{attribute 'linkalways'} 
{attribute 'no_explicit_call' := 'This FB is a CLASS and must be accessed using methods or properties'}
FUNCTION_BLOCK Nci EXTENDS CyclicInstance IMPLEMENTS I_Nci
VAR
	_nciPlc : NciPlc;
END_VAR

PROPERTY _InternalNciPlcRef : REFERENCE TO NciPlc
GET
_InternalNciPlcRef REF= _nciPlc;
END_GET
END_PROPERTY

METHOD AddAxisToGroup
VAR_INPUT
	axis : I_Axis;
	index : UDINT;
	timeout : TIME;
	feedback : REFERENCE TO I_CommandFeedback;
END_VAR
VAR_INST
	pCmd : POINTER TO AddAxisToGroupCommand;
END_VAR
VAR
	_axis : I_Axis;
	_index : UDINT;
	_timeout : TIME;
END_VAR
_axis := axis;
_index := index;
_timeout := timeout;

pCmd := __NEW(AddAxisToGroupCommand(
	nci := THIS^,
	axis := _axis,
	index := _index,
	timeout := _timeout
));

(*
This doesn't work hence the horrible hack with intermediate values

pCmd := __NEW(AddAxisToGroupCommand(
	nci := THIS^,
	axis := axis,
	index := index,
	timeout := timeout
));
*)

pCmd^.Execute(feedback).ThenRelease();
END_METHOD

PROPERTY BlockNumber : UDINT
GET
BlockNumber := ItpGetBlockNumber(THIS^._nciPlc.nciToPlc);
END_GET
END_PROPERTY

METHOD BuildXYGroup
VAR_INPUT
	xAxis : I_Axis;
	yAxis : I_Axis;
	timeout : TIME;
	feedback : REFERENCE TO I_CommandFeedback;
END_VAR
VAR
	null : I_Axis;
END_VAR
BuildXYZGroup(xAxis, yAxis, null, timeout, feedback);
END_METHOD

METHOD BuildXYZGroup
VAR_INPUT
	xAxis : I_Axis;
	yAxis : I_Axis;
	zAxis : I_Axis;
	timeout : TIME;
	feedback : REFERENCE TO I_CommandFeedback;
END_VAR
VAR_INST
	pCmd : POINTER TO BuildXYZGroupCommand;
END_VAR
VAR
	_xAxis : I_Axis;
	_yAxis : I_Axis;
	_zAxis : I_Axis;
	_timeout : TIME;
END_VAR
_xAxis := xAxis;
_yAxis := yAxis;
_zAxis := zAxis;
_timeout := timeout;

pCmd := __NEW(BuildXYZGroupCommand(
	nci := THIS^,
	xAxis := _xAxis,
	yAxis := _yAxis,
	zAxis := _zAxis,
	timeout := _timeout
));

(*
This doesn't work hence the horrible hack with intermediate values

pCmd := __NEW(BuildXYZGroupCommand(
	nci := THIS^,
	xAxis := xAxis,
	yAxis := yAxis,
	zAxis := zAxis,
	timeout := commandTimeout
));
*)

pCmd^.Execute(feedback).ThenRelease();
END_METHOD

PROPERTY ChannelId : UINT
GET
ChannelId := ItpGetChannelId(THIS^._nciPlc.nciToPlc);
END_GET
END_PROPERTY

PROPERTY ChannelType : ChannelType
GET
VAR
	inter : INT;
	pInter : POINTER TO ChannelType;
END_VAR
// Don't know how to do the type conversion with NCIChannelType being strict
inter := ItpGetChannelType(THIS^._nciPlc.nciToPlc);
pInter := ADR(inter);
ChannelType := pInter^;
END_GET
END_PROPERTY

METHOD  CyclicCall
END_METHOD

PROPERTY ErrorId : UDINT
GET
ErrorId := ItpGetError(THIS^._nciPlc.nciToPlc);
END_GET
END_PROPERTY

METHOD GetGroupAxisIds : DWORD
VAR_IN_OUT
	axisIds : ARRAY[1..8] OF DWORD;
END_VAR
GetGroupAxisIds := ItpGetGroupAxisIds(axisIds, THIS^._nciPlc.nciToPlc);
END_METHOD

METHOD GetOverride : LREAL
GetOverride := ItpGetOverridePercent(THIS^._nciPlc.plcToNci);
END_METHOD

PROPERTY GroupId : UDINT
GET
GroupId := ItpGetGroupId(THIS^._nciPlc.nciToPlc);
END_GET
END_PROPERTY

PROPERTY HandshakeableMFunction : INT
GET
HandshakeableMFunction := ItpGetHskMFunc(THIS^._nciPlc.nciToPlc);
END_GET
END_PROPERTY

PROPERTY HasError : BOOL
GET
HasError := ItpHasError(THIS^._nciPlc.nciToPlc);
END_GET
END_PROPERTY

PROPERTY HParam : DINT
GET
HParam := ItpGetHParam(THIS^._nciPlc.nciToPlc);
END_GET
END_PROPERTY

PROPERTY InterpreterState : UDINT
GET
InterpreterState := ItpGetStateInterpreter(THIS^._nciPlc.nciToPlc);
END_GET
END_PROPERTY

PROPERTY IsEstop : BOOL
GET
IsEstop := ItpIsEStopEx(THIS^._nciPlc.nciToPlc);
END_GET
END_PROPERTY

METHOD IsFastMFunctionPresent : BOOL
VAR_INPUT
	functionNumber : INT;
END_VAR
IsFastMFunctionPresent := ItpIsFastMFunc(functionNumber, THIS^._nciPlc.nciToPlc);
END_METHOD

METHOD IsHandshakeableMFunctionPresent : BOOL
IsHandshakeableMFunctionPresent := ItpIsHskMFunc(THIS^._nciPlc.nciToPlc);
END_METHOD

METHOD ReadCyclicLRealParameter : LREAL
VAR_INPUT
	parameterNumber : UINT(1..4);
END_VAR
CASE parameterNumber OF
	1: ReadCyclicLRealParameter := ItpReadCyclicLRealParam1(THIS^._nciPlc.nciToPlc);
	2: ReadCyclicLRealParameter := ItpReadCyclicLRealParam2(THIS^._nciPlc.nciToPlc);
	3: ReadCyclicLRealParameter := ItpReadCyclicLRealParam3(THIS^._nciPlc.nciToPlc);
	4: ReadCyclicLRealParameter := ItpReadCyclicLRealParam4(THIS^._nciPlc.nciToPlc);
END_CASE
END_METHOD

METHOD ReadCyclicUdintParameter : UDINT
VAR_INPUT
	parameterNumber : UINT(1..4);
END_VAR
CASE parameterNumber OF
	1: ReadCyclicUdintParameter := ItpReadCyclicUdintParam1(THIS^._nciPlc.nciToPlc);
	2: ReadCyclicUdintParameter := ItpReadCyclicUdintParam2(THIS^._nciPlc.nciToPlc);
	3: ReadCyclicUdintParameter := ItpReadCyclicUdintParam3(THIS^._nciPlc.nciToPlc);
	4: ReadCyclicUdintParameter := ItpReadCyclicUdintParam4(THIS^._nciPlc.nciToPlc);
END_CASE
END_METHOD

METHOD ReleaseAxis
VAR_INPUT
	axis : I_Axis;
	timeout : TIME;
	feedback : REFERENCE TO I_CommandFeedback;
END_VAR
VAR_INST
	pCmd : POINTER TO ReleaseAxisCommand;
END_VAR
VAR
	_axis : I_Axis;
	_timeout : TIME;
END_VAR
_axis := axis;
_timeout := timeout;

pCmd := __NEW(ReleaseAxisCommand(
	axis := _axis,
	timeout := _timeout
));

(*
This doesn't work hence the horrible hack with intermediate values

pCmd := __NEW(ReleaseAxisCommand(
	axis := axis,
	timeout := timeout
));
*)
pCmd^.Execute(feedback).ThenRelease();
END_METHOD

METHOD ResetGroup
VAR_INPUT
	timeout : TIME;
	feedback : REFERENCE TO I_CommandFeedback;
END_VAR
VAR_INST
	pCmd : POINTER TO ResetGroupCommand;
END_VAR
VAR
	_timeout : TIME;
END_VAR
_timeout := timeout;

pCmd := __NEW(ResetGroupCommand(
	nci := THIS^,
	timeout := _timeout
));

(*
This doesn't work hence the horrible hack with intermediate values

pCmd := __NEW(ResetGroupCommand(
	nci := THIS^,
	timeout := timeout
));
*)

pCmd^.Execute(feedback).ThenRelease();
END_METHOD

METHOD SetOverride : BOOL
VAR_INPUT
	value : LREAL;
END_VAR
SetOverride := ItpSetOverridePercent(value, THIS^._nciPlc.plcToNci);
END_METHOD

PROPERTY SetPathVelocity : LREAL
GET
SetPathVelocity := ItpGetSetPathVelocity(THIS^._nciPlc.nciToPlc);
END_GET
END_PROPERTY

PROPERTY SParam : UINT
GET
SParam := ItpGetSParam(THIS^._nciPlc.nciToPlc);
END_GET
END_PROPERTY

PROPERTY TParam : UINT
GET
TParam := ItpGetTParam(THIS^._nciPlc.nciToPlc);
END_GET
END_PROPERTY

END_FUNCTION_BLOCK

(* stored: Version 1.1.0.1, ProductVersion 3.1.4024.12
   POU Nci: Id {f4f57f23-d325-0909-0740-6ef1501e4700}, SpecialFunc None
   Folder Configuration: Id {88eb77e5-8505-0b13-208d-06ae6cb833ec}
   Folder Internal Properties: Id {5c441f11-5c36-4a25-a469-77832f6c3ab5}
   Folder Methods: Id {eb3c7eaf-dfb5-0372-0016-cb165d65c918}
   Folder Properties: Id {9b308d9c-cf3d-093c-3584-5ad4df15e20d}
   Property _InternalNciPlcRef: Id {09415743-66c1-434a-b941-e21d020bb5bf}
   Get Get: Id {949a3851-8449-45a9-892f-a26cda235f58}
   Method AddAxisToGroup: Id {5d45a9a7-6d05-0d2b-27b5-79ba5b2eb2c7}
   Property BlockNumber: Id {ed372b87-29b3-0a1a-0b74-a10370d405f8}
   Get Get: Id {f93c51fc-0941-0b17-1306-659017cf0a9e}
   Method BuildXYGroup: Id {9849a2df-cafa-0395-3040-8d89f7219b15}
   Method BuildXYZGroup: Id {d4df4ca0-a512-0b57-3ad2-c0cda1e1758d}
   Property ChannelId: Id {09b3ab1e-9925-01cb-30ce-90054bf786f8}
   Get Get: Id {b6a23344-1051-0c06-1d5e-15387b416b28}
   Property ChannelType: Id {d49fd91a-aca9-0237-2591-75a0198a0fa3}
   Get Get: Id {d55f81ea-7033-0dd4-2311-969f8baef65a}
   Method CyclicCall: Id {838887cb-7f06-09de-3df5-bf0a2be36fcc}
   Property ErrorId: Id {f369e32b-cc56-0313-12c3-ecf9c674699a}
   Get Get: Id {82008dd1-ebe7-0696-160f-5c73506db06e}
   Method GetGroupAxisIds: Id {f7a6d126-e2b6-0bc6-3a4d-c5d6738f9962}
   Method GetOverride: Id {58a4283c-4b05-0d2c-31b9-e1ff0c76c9f9}
   Property GroupId: Id {e0517028-3a9d-026a-385e-bb8ac1a641ff}
   Get Get: Id {1e32072f-7668-0272-02e1-9e42282c0086}
   Property HandshakeableMFunction: Id {8c10b698-bef7-04d2-3038-563b4f835b24}
   Get Get: Id {f652a4d7-1be6-0813-2d9f-e4a827a80355}
   Property HasError: Id {9263d7f0-3daa-0052-0803-c5e977270099}
   Get Get: Id {55a3aeeb-4e6b-0ba1-1f66-c461721621fd}
   Property HParam: Id {d73b387f-5953-0d9f-35c1-153b9d3dd768}
   Get Get: Id {a22b731f-839f-0871-3aee-c7b6cb2aee37}
   Property InterpreterState: Id {57655ad1-7d01-0963-122c-3c0563f86dc5}
   Get Get: Id {0088775a-c1e4-0e2e-368b-b3d2d41914a6}
   Property IsEstop: Id {96e5e85e-3ad3-0eca-0c9c-5fbe002bf275}
   Get Get: Id {233bff47-1521-030d-10bc-d381218d2a38}
   Method IsFastMFunctionPresent: Id {5732f7c0-a406-0419-3cac-84082892815a}
   Method IsHandshakeableMFunctionPresent: Id {a0aa6003-b6a8-0bc9-0a46-c04aaee12e44}
   Method ReadCyclicLRealParameter: Id {ac0a4f2b-e74e-05a9-1ba2-7e50dbd409c9}
   Method ReadCyclicUdintParameter: Id {e83684d5-4fdf-0d03-343e-dff776ded206}
   Method ReleaseAxis: Id {85630d2c-a95a-07c1-0581-d3d81b1fea01}
   Method ResetGroup: Id {5a4cbab8-254e-0c2f-3388-108e0e893560}
   Method SetOverride: Id {ff5194d3-333b-0a27-00d0-c5c7f97bb8c5}
   Property SetPathVelocity: Id {f2a4b773-26ea-0bc8-160f-854fdb045118}
   Get Get: Id {5fc7a4ac-330b-09a8-0c99-cb103ef06c27}
   Property SParam: Id {cd33a989-617f-0769-2aaa-454de48eef34}
   Get Get: Id {8db5b9d4-d342-0a82-2573-ba894df90968}
   Property TParam: Id {cde84c08-7c26-0d10-322b-8c504543b0d6}
   Get Get: Id {23b4bd45-55ff-098b-30a0-b2f28dae9e2e} *)
